FUNCTION_BLOCK Ventilation EXTENDS Device IMPLEMENTS SHLib.IOutputDevice
VAR
	_Speed : BYTE;
END_VAR

{attribute 'monitoring' := 'call'}
PROPERTY IsOn : BOOL
GET
IsOn := _Speed <> 0;
END_GET
END_PROPERTY

{attribute 'monitoring' := 'call'}
PROPERTY Name : STRING
GET
Name := 'Ventilation';
END_GET
END_PROPERTY

METHOD SetSpeed
VAR_INPUT
	speed : BYTE;
END_VAR
_Speed := speed;
END_METHOD

{attribute 'monitoring' := 'call'}
PROPERTY Speed : BYTE
GET
Speed := _Speed;
END_GET
END_PROPERTY

METHOD WriteOutputs
// put values to terminal here
END_METHOD

END_FUNCTION_BLOCK

(* stored: Version 1.1.0.1
   POU Ventilation: Id {519c61d9-5da5-47c5-aef5-3169a8420acb}, SpecialFunc None
   Property IsOn: Id {b650a8dd-aa93-4f9b-8d25-25094f09fbcf}
   Get Get: Id {64fc3015-fa56-47bd-a048-8496cfec0747}
   Property Name: Id {4177a6ae-2fb0-4458-a816-f09274b12068}
   Get Get: Id {b9e238b8-1989-441a-907c-43e20a23d556}
   Method SetSpeed: Id {783ccaf6-9e73-4bc7-bd32-16c93365334b}
   Property Speed: Id {611a69b3-a767-49a8-aa02-6ce0ae25f464}
   Get Get: Id {0d0dfc88-2384-4a83-b468-fffe19243b1e}
   Method WriteOutputs: Id {195de019-3db1-4311-8214-fb1ef64b03ce} *)
